KUKA KRL program: Eingabe.src, Eingabe.dat

--- Eingabe.src ---
&ACCESS RVO1
&COMMENT
DEF Eingabe ( )
;FOLD INI
  ;FOLD BASISTECH INI
    GLOBAL INTERRUPT DECL 3 WHEN $STOPMESS==TRUE DO IR_STOPM ( )
    INTERRUPT ON 3
    BAS (#INITMOV,0 )
  ;ENDFOLD (BASISTECH INI)
  ;FOLD USER INI
    ;Make your modifications here

  ;ENDFOLD (USER INI)
;ENDFOLD (INI)

;FOLD PTP HOME  Vel= 100 % DEFAULT;%{PE}%MKUKATPBASIS,%CMOVE,%VPTP,%P 1:PTP, 2:HOME, 3:, 5:100, 7:DEFAULT
$BWDSTART = FALSE
PDAT_ACT=PDEFAULT
FDAT_ACT=FHOME
BAS (#PTP_PARAMS,100 )
$H_POS=XHOME
PTP  XHOME
;ENDFOLD
MsgDialog(zeile,"Zeile eingeben",,,"3", "2", "1")
MsgDialog(spalte,"Spalte eingeben",,,"3", "2", "1")
MsgNotify("Zeile: %1", "Test", zeile)
MsgNotify("Spalte: %1", "Test", spalte)



zeile = zeile - 5
spalte = spalte - 5

xkoord = spalte * seitenlaenge
ykoord = zeile * seitenlaenge

MsgNotify("xkoord: %1", "Test", xkoord)
MsgNotify("ykoord: %1", "Test", ykoord)

cur = base
cur.X = cur.X + xkoord
cur.Y = cur.Y + ykoord
cur.Z = cur.Z - 10

;FOLD PTP cur  Vel=100 % PDAT2 Tool[15] Base[15];%{PE}%R 8.3.22,%MKUKATPBASIS,%CMOVE,%VPTP,%P 1:PTP, 2:cur, 3:, 5:100, 7:PDAT2
$BWDSTART=FALSE
PDAT_ACT=PPDAT2
FDAT_ACT=Fcur
BAS(#PTP_PARAMS,100)
PTP Xcur
;ENDFOLD

cur.Z = base.Z
;FOLD PTP cur  Vel=100 % PDAT2 Tool[15] Base[15];%{PE}%R 8.3.22,%MKUKATPBASIS,%CMOVE,%VPTP,%P 1:PTP, 2:cur, 3:, 5:100, 7:PDAT2
$BWDSTART=FALSE
PDAT_ACT=PPDAT2
FDAT_ACT=Fcur
BAS(#PTP_PARAMS,100)
PTP Xcur
;ENDFOLD

; draw

cur.Z = base.Z - 10
;FOLD PTP cur  Vel=100 % PDAT2 Tool[15] Base[15];%{PE}%R 8.3.22,%MKUKATPBASIS,%CMOVE,%VPTP,%P 1:PTP, 2:cur, 3:, 5:100, 7:PDAT2
$BWDSTART=FALSE
PDAT_ACT=PPDAT2
FDAT_ACT=Fcur
BAS(#PTP_PARAMS,100)
PTP Xcur
;ENDFOLD

WAIT SEC 2
;FOLD PTP HOME  Vel= 100 % DEFAULT;%{PE}%MKUKATPBASIS,%CMOVE,%VPTP,%P 1:PTP, 2:HOME, 3:, 5:100, 7:DEFAULT
$BWDSTART = FALSE
PDAT_ACT=PDEFAULT
FDAT_ACT=FHOME
BAS (#PTP_PARAMS,100 )
$H_POS=XHOME
PTP  XHOME
;ENDFOLD

END

--- Eingabe.dat ---
&ACCESS RVO1
&COMMENT
DEFDAT Eingabe PUBLIC
;FOLD EXTERNAL DECLARATIONS;%{PE}%MKUKATPBASIS,%CEXT,%VCOMMON,%P
;FOLD BASISTECH EXT;%{PE}%MKUKATPBASIS,%CEXT,%VEXT,%P
EXT  BAS (BAS_COMMAND  :IN,REAL  :IN )
DECL INT SUCCESS
;ENDFOLD (BASISTECH EXT)
;FOLD USER EXT;%{E}%MKUKATPUSER,%CEXT,%VEXT,%P
;Make here your modifications

;ENDFOLD (USER EXT)
;ENDFOLD (EXTERNAL DECLERATIONS)
DECL INT zeile
DECL INT spalte
DECL INT xkoord
DECL INT ykoord
DECL INT seitenlaenge = 100
DECL E6POS base = {X 0, Y 0, Z 0, A 0, B 0, C 0}
DECL E6POS cur
DECL E6POS Xbase={X 0,Y 0,Z 0,A 0,B 0,C 0,S 0,T 0,E1 0,E2 0,E3 0,E4 0,E5 0,E6 0}
DECL FDAT Fbase={TOOL_NO 0,BASE_NO 0,IPO_FRAME #BASE,POINT2[] " ",TQ_STATE FALSE}
DECL PDAT PPDAT0={VEL 1,ACC 100,APO_DIST 100,APO_MODE #CPTP,GEAR_JERK 50}
DECL BASIS_SUGG_T LAST_BASIS={POINT1[] "base",POINT2[] "base",CP_PARAMS[] "CPDAT9",PTP_PARAMS[] "PDAT2",CONT[] " ",CP_VEL[] "1",PTP_VEL[] "100",SYNC_PARAMS[] "SYNCDAT ",SPL_NAME[] "S0 "}
DECL PDAT PPDAT2={VEL 100,ACC 100,APO_DIST 100,APO_MODE #CPTP,GEAR_JERK 50}
DECL E6POS Xcur={X 0,Y 0,Z 0,A 0,B 0,C 0,S 0,T 0,E1 0,E2 0,E3 0,E4 0,E5 0,E6 0}
DECL FDAT Fcur={TOOL_NO 0,BASE_NO 0,IPO_FRAME #BASE,POINT2[] " ",TQ_STATE FALSE}
ENDDAT
